{attribute 'linkalways'} 
{attribute 'no_explicit_call' := 'This FB is a CLASS and must be accessed using methods or properties'}
{attribute 'enable_dynamic_creation'}
FUNCTION_BLOCK FINAL MOD_LREAL EXTENDS Node
VAR
	in1 : _LREAL(0.0);
	in2 : _LREAL(0.0);
	out : _LREAL(0.0);
END_VAR

METHOD PUBLIC Clone : I_Node
VAR
	pNode : POINTER TO MOD_LREAL;
END_VAR
pNode := __NEW(MOD_LREAL);
Clone := pNode^;
END_METHOD

METHOD FB_init : BOOL
VAR_INPUT
	bInitRetains : BOOL; // if TRUE, the retain variables are initialized (warm start / cold start)
	bInCopyCode : BOOL;  // if TRUE, the instance afterwards gets moved into the copy code (online change)
END_VAR
AddInput('in1',THIS^.in1);
AddInput('in2',THIS^.in2);
AddOutput('out', THIS^.out);
END_METHOD

METHOD PROTECTED OnExecute
VAR
END_VAR
out.Value := LMOD(in1.Value, in2.Value);
END_METHOD

END_FUNCTION_BLOCK

(* stored: Version 1.1.0.1, ProductVersion 3.1.4024.15
   POU MOD_LREAL: Id {8deb97e4-b4cd-41e0-8254-4a76a1f4019f}, SpecialFunc None
   Folder Constructor: Id {c02f8ebb-6def-4949-aa67-5905f9623d64}
   Method Clone: Id {18ce49cd-aeb1-488c-897b-46e2febb04b9}
   Method FB_init: Id {0e803b7f-17cd-4d1d-ad88-8af3617233a3}
   Method OnExecute: Id {32f46c1b-c96d-4b90-9e53-bb79c3010f2c} *)
